// TIA Portal V17 export
// export: Created 2024-09-02T12:50:24.0315334Z, ExportSetting WithDefaults, DisplayName Totally Integrated Automation Portal, DisplayVersion V17, DisplayName TIA Portal Openness, DisplayVersion V17, DisplayName TIA Portal Version Control Interface, DisplayVersion V17, DisplayName STEP 7 Professional, DisplayVersion V17, DisplayName STEP 7 Safety, DisplayVersion V17, DisplayName WinCC Professional, DisplayVersion V17
DATA_BLOCK "DB_MES_CONT_INTERFACE_OP70"   // DB700
{ S7_Optimized_Access := 'FALSE' }
VERSION : 0.1
// stored: AutoNumber false, DBAccessibleFromOPCUA true, IsOnlyStoredInLoadMemory false, IsWriteProtectedInAS false
   VAR
      c : Byte;   // %X0 - (WS)Media ON, %X1 - (WS)Hand selected, %X2 - (WS)Auto selected, %X3 -(WS)Start ON(with auto or hand Mode), %X4 -(WS)Error, %X5 - (WS)Clock_1Hz - lifebit, %X6 -(MES)Clock_1Hz - lifebit , %X7 - (MES)Automatic on Conveyor
      Really_Time_Status_OP70_2 : Byte;   // %X0 - (WS)Media ON, %X1 - (WS)Hand selected, %X2 - (WS)Auto selected, %X3 -(WS)Start ON(with auto or hand Mode), %X4 -(WS)Error, %X5 - (WS)Clock_1Hz - lifebit, %X6 -(MES)Clock_1Hz - lifebit , %X7 - (MES)Automatic on Conveyor
      Really_Time_Status_OP70_3 : Byte;   // %X0 - (WS)Media ON, %X1 - (WS)Hand selected, %X2 - (WS)Auto selected, %X3 -(WS)Start ON(with auto or hand Mode), %X4 -(WS)Error, %X5 - (WS)Clock_1Hz - lifebit, %X6 -(MES)Clock_1Hz - lifebit , %X7 - (MES)Automatic on Conveyor
      Start_Comunication_Reading_OP70_1 { ExternalAccessible := 'False'; ExternalVisible := 'False'; ExternalWritable := 'False'} : Bool;
      Start_Comunication_Reading_OP70_2 { ExternalAccessible := 'False'; ExternalVisible := 'False'; ExternalWritable := 'False'} : Bool;
      Start_Comunication_Reading_OP70_3 { ExternalAccessible := 'False'; ExternalVisible := 'False'; ExternalWritable := 'False'} : Bool;
      Start_Comunication_Saving_OP70_1 { ExternalAccessible := 'False'; ExternalVisible := 'False'; ExternalWritable := 'False'} : Bool;
      Start_Comunication_Saving_OP70_2 { ExternalAccessible := 'False'; ExternalVisible := 'False'; ExternalWritable := 'False'} : Bool;
      Start_Comunication_Saving_OP70_3 { ExternalAccessible := 'False'; ExternalVisible := 'False'; ExternalWritable := 'False'} : Bool;
      Done_Reading_OP70_1 : Bool;
      Done_Saving_OP70_1 : Bool;
      Done_Reading_OP70_2 : Bool;
      Done_Saving_OP70_2 : Bool;
      Done_Reading_OP70_3 : Bool;
      Done_Saving_OP70_3 : Bool;
      WS_ReallyTime : Struct
         "Counter" : IEC_COUNTER;
         PLC_Alive { S7_SetPoint := 'True'} : Int;
      END_STRUCT;
      Concentrator_ReallyTime : Struct
         Concentrator_Alive : Int;
         Old_WordLife : Int;
         Error_inCommunication : Bool;
      END_STRUCT;
   END_VAR
BEGIN
END_DATA_BLOCK
